// TIA Portal project "plc作业" (V15.1)

(* hardware
DEVICE "HMI_1"  KTP700 Basic PN
   slot 0: "HMI_1"  KTP700 Basic PN  6AV2 123-2GB03-0AX0  15.1.0.0
   slot 1: "HMI_RT_1"  KTP700 Basic PN  6AV2 123-2GB03-0AX0  15.1.0.0
   slot 5: "HMI_1.IE_CP_1"  PROFINET Interface  15.0.1.0
      slot 1: "PROFINET Interface_1"  PROFINET Interface
         slot 1: "Port_1"  Port
DEVICE "S7-1200 station_1"  S7-1200 Station
   slot 0: "Rack_0"  S7-1200 Rack  Rack  V1.0
   slot 1: "PLC_1"  CPU 1214C DC/DC/DC  6ES7 214-1AG40-0XB0  V4.2
*)

// ===== PLC "PLC_1"  CPU 1214C DC/DC/DC =====

VAR_GLOBAL   // PLC tag table "默认变量表"
   "Tag_1" AT %M500.0 : Bool;
   "Tag_2" AT %M500.1 : Bool;
   "Tag_3" AT %M500.2 : Bool;
   "Tag_22" AT %M501.0 : Bool;
   "Tag_23" AT %M501.1 : Bool;
   "Tag_24" AT %M501.2 : Bool;
   "Tag_25" AT %M500.5 : Bool;
   "Tag_26" AT %M500.6 : Bool;
   "Tag_27" AT %M500.7 : Bool;
END_VAR

VAR_GLOBAL   // PLC tag table "左车道检测"
   "使能信号" AT %I0.6 : Bool;
   "左车道入口计数" AT %I0.7 : Bool;
   "左车道出口计数" AT %I1.1 : Bool;
   "左车道计数清零" AT %I1.3 : Bool;
   "左车道封闭" AT %Q0.2 : Bool;
   "左车道堵塞" AT %Q0.3 : Bool;
   "左车道拥堵" AT %Q0.4 : Bool;
   "左车道畅通" AT %Q0.5 : Bool;
   "左车道hmi停止控制" AT %M2.0 : Bool;
   "左车道错误" AT %M2.1 : Bool;
END_VAR

VAR_GLOBAL   // PLC tag table "右车道"
   "右车道入口计数" AT %I1.0 : Bool;
   "右车道出口计数" AT %I1.2 : Bool;
   "右车道计数清零" AT %I1.4 : Bool;
   "右车道封闭" AT %Q0.6 : Bool;
   "右车道堵塞" AT %Q0.7 : Bool;
   "右车道拥堵" AT %Q1.0 : Bool;
   "右车道畅通" AT %Q1.1 : Bool;
   "右车道hmi停止控制" AT %M2.2 : Bool;
   "右车道错误" AT %M2.3 : Bool;
END_VAR

DATA_BLOCK "车辆检测_DB"   // DB1
{ S7_Optimized_Access := 'FALSE' }
VERSION : 0.1
// stored: InstanceOfName 车辆检测
"车辆检测"
BEGIN
   堵塞设定数量 := 15;
   拥堵设定数量 := 10;
END_DATA_BLOCK

DATA_BLOCK "车辆检测_DB_1"   // DB2
{ S7_Optimized_Access := 'FALSE' }
VERSION : 0.1
// stored: InstanceOfName 车辆检测
"车辆检测"
BEGIN
   堵塞设定数量 := 15;
   拥堵设定数量 := 10;
END_DATA_BLOCK

FUNCTION_BLOCK "车辆检测"   // FB1, LAD
{ S7_Optimized_Access := 'FALSE' }
VERSION : 0.1
   VAR_INPUT
      使能信号 : Bool;
      车道入口计数 : Bool;
      出口计数 : Bool;
      计数清零 : Bool;
      停止控制 : Bool;
   END_VAR
   VAR_OUTPUT
      封闭 : Bool;
      堵塞 : Bool;
      拥堵 : Bool;
      畅通 : Bool;
      错误 : Bool;
   END_VAR
   VAR_IN_OUT
      堵塞设定数量 : Int;
      拥堵设定数量 : Int;
      当前车辆数量 : Int;
      "step" : Bool;
   END_VAR
   VAR_TEMP   // added for the SCL form of the ladder/FBD networks
      _w1 : Bool;
      _w2 : Bool;
   END_VAR
BEGIN

REGION Network 1
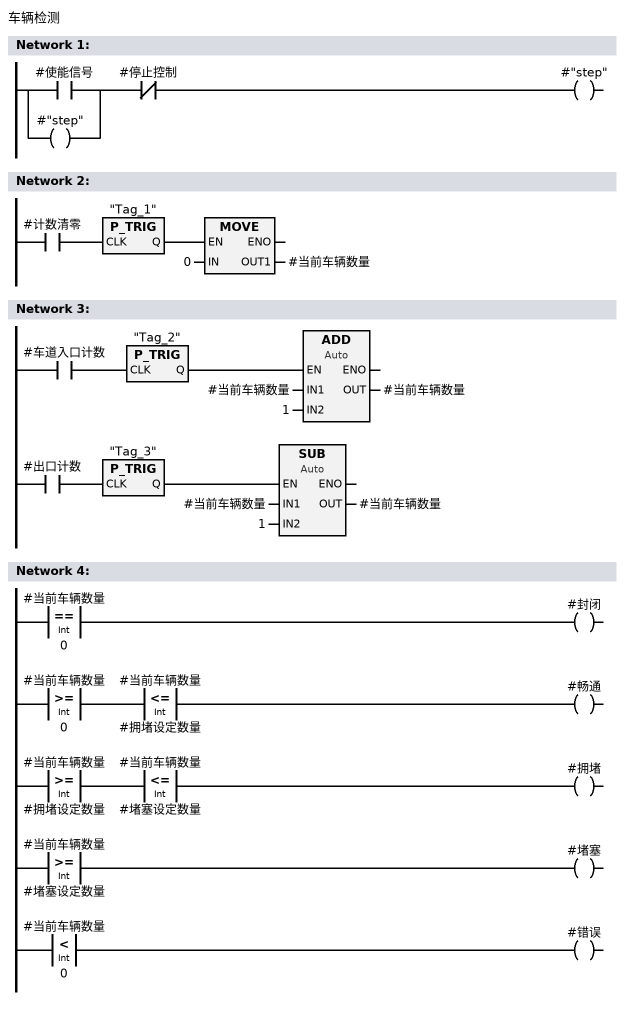
   RUNG wire#powerrail
      Contact( #使能信号 )
      wire#w1
      I_Contact( #停止控制 )
      Coil( #"step" )
   END_RUNG
   RUNG wire#powerrail
      Coil( #"step" )
   END_RUNG wire#w1
   // the same network as SCL:
   #"step" := TRUE;
   #"step" := (#使能信号 OR TRUE) AND NOT #停止控制;
END_REGION

REGION Network 2
   RUNG wire#powerrail
      Contact( #计数清零 )
      P_Trig( "Tag_1" )
      Move(in := 0, out1 => #当前车辆数量)
   END_RUNG
   // the same network as SCL:
   #_w1 := #计数清零 AND NOT "Tag_1";   // rising edge
   "Tag_1" := #计数清零;
   IF #_w1 THEN #当前车辆数量 := 0; END_IF;
END_REGION

REGION Network 3
   RUNG wire#powerrail
      Contact( #车道入口计数 )
      P_Trig( "Tag_2" )
      Add(in1 := #当前车辆数量, in2 := 1, out => #当前车辆数量)
   END_RUNG
   RUNG wire#powerrail
      Contact( #出口计数 )
      P_Trig( "Tag_3" )
      Sub(in1 := #当前车辆数量, in2 := 1, out => #当前车辆数量)
   END_RUNG
   // the same network as SCL:
   #_w1 := #车道入口计数 AND NOT "Tag_2";   // rising edge
   "Tag_2" := #车道入口计数;
   IF #_w1 THEN #当前车辆数量 := #当前车辆数量 + 1; END_IF;
   #_w2 := #出口计数 AND NOT "Tag_3";   // rising edge
   "Tag_3" := #出口计数;
   IF #_w2 THEN #当前车辆数量 := #当前车辆数量 - 1; END_IF;
END_REGION

REGION Network 4
   RUNG wire#powerrail
      { S7_Templates := "SrcType := Int" } EQ_Contact(in1 := #当前车辆数量, in2 := 0)
      Coil( #封闭 )
   END_RUNG
   RUNG wire#powerrail
      { S7_Templates := "SrcType := Int" } GE_Contact(in1 := #当前车辆数量, in2 := 0)
      { S7_Templates := "SrcType := Int" } LE_Contact(in1 := #当前车辆数量, in2 := #拥堵设定数量)
      Coil( #畅通 )
   END_RUNG
   RUNG wire#powerrail
      { S7_Templates := "SrcType := Int" } GE_Contact(in1 := #当前车辆数量, in2 := #拥堵设定数量)
      { S7_Templates := "SrcType := Int" } LE_Contact(in1 := #当前车辆数量, in2 := #堵塞设定数量)
      Coil( #拥堵 )
   END_RUNG
   RUNG wire#powerrail
      { S7_Templates := "SrcType := Int" } GE_Contact(in1 := #当前车辆数量, in2 := #堵塞设定数量)
      Coil( #堵塞 )
   END_RUNG
   RUNG wire#powerrail
      { S7_Templates := "SrcType := Int" } LT_Contact(in1 := #当前车辆数量, in2 := 0)
      Coil( #错误 )
   END_RUNG
   // the same network as SCL:
   #封闭 := #当前车辆数量 = 0;
   #畅通 := (#当前车辆数量 >= 0) AND (#当前车辆数量 <= #拥堵设定数量);
   #拥堵 := (#当前车辆数量 >= #拥堵设定数量) AND (#当前车辆数量 <= #堵塞设定数量);
   #堵塞 := #当前车辆数量 >= #堵塞设定数量;
   #错误 := #当前车辆数量 < 0;
END_REGION
END_FUNCTION_BLOCK

ORGANIZATION_BLOCK "Main"   // OB1, LAD, ProgramCycle
TITLE = "Main Program Sweep (Cycle)"
{ S7_Optimized_Access := 'TRUE' }
VERSION : 0.1
   VAR_INPUT
      Initial_Call : Bool;   // Initial call of this OB
      Remanence : Bool;   // =True, if remanent data are available
   END_VAR
   VAR_TEMP   // added for the SCL form of the ladder/FBD networks
      _w1 : Bool;
      _w2 : Bool;
      _w3 : Bool;
   END_VAR
BEGIN

REGION Network 1: 左车道
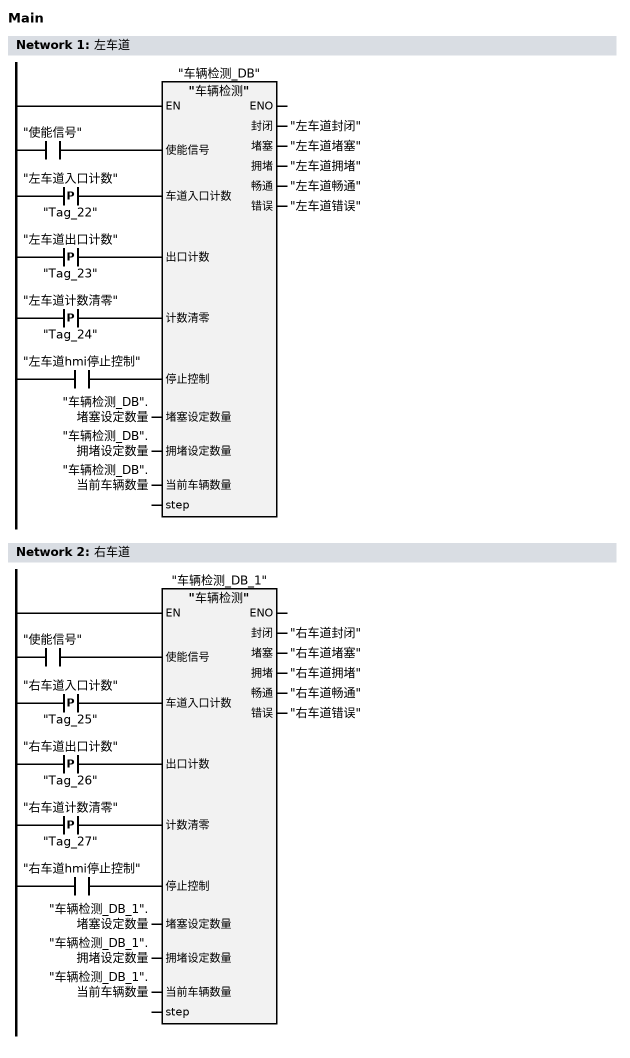
   RUNG wire#powerrail
      "车辆检测_DB"(使能信号 := wire#w1, 车道入口计数 := wire#w2, 出口计数 := wire#w3, 计数清零 := wire#w4, 停止控制 := wire#w5, 堵塞设定数量 := "车辆检测_DB".堵塞设定数量, 拥堵设定数量 := "车辆检测_DB".拥堵设定数量, 当前车辆数量 := "车辆检测_DB".当前车辆数量, "step" :=, 封闭 => "左车道封闭", 堵塞 => "左车道堵塞", 拥堵 => "左车道拥堵", 畅通 => "左车道畅通", 错误 => "左车道错误")
   END_RUNG
   RUNG wire#powerrail
      Contact( "使能信号" )
   END_RUNG wire#w1
   RUNG wire#powerrail
      P_Contact(operand := "左车道入口计数", bit := "Tag_22")
   END_RUNG wire#w2
   RUNG wire#powerrail
      P_Contact(operand := "左车道出口计数", bit := "Tag_23")
   END_RUNG wire#w3
   RUNG wire#powerrail
      P_Contact(operand := "左车道计数清零", bit := "Tag_24")
   END_RUNG wire#w4
   RUNG wire#powerrail
      Contact( "左车道hmi停止控制" )
   END_RUNG wire#w5
   // the same network as SCL:
   #_w1 := "左车道入口计数" AND NOT "Tag_22";   // rising edge of "左车道入口计数"
   "Tag_22" := "左车道入口计数";
   #_w2 := "左车道出口计数" AND NOT "Tag_23";   // rising edge of "左车道出口计数"
   "Tag_23" := "左车道出口计数";
   #_w3 := "左车道计数清零" AND NOT "Tag_24";   // rising edge of "左车道计数清零"
   "Tag_24" := "左车道计数清零";
   "车辆检测_DB"(使能信号 := "使能信号",   // "车辆检测"
             车道入口计数 := #_w1,
             出口计数 := #_w2,
             计数清零 := #_w3,
             停止控制 := "左车道hmi停止控制",
             堵塞设定数量 := "车辆检测_DB".堵塞设定数量,
             拥堵设定数量 := "车辆检测_DB".拥堵设定数量,
             当前车辆数量 := "车辆检测_DB".当前车辆数量,
             封闭 => "左车道封闭",
             堵塞 => "左车道堵塞",
             拥堵 => "左车道拥堵",
             畅通 => "左车道畅通",
             错误 => "左车道错误");
END_REGION

REGION Network 2: 右车道
   RUNG wire#powerrail
      "车辆检测_DB_1"(使能信号 := wire#w1, 车道入口计数 := wire#w2, 出口计数 := wire#w3, 计数清零 := wire#w4, 停止控制 := wire#w5, 堵塞设定数量 := "车辆检测_DB_1".堵塞设定数量, 拥堵设定数量 := "车辆检测_DB_1".拥堵设定数量, 当前车辆数量 := "车辆检测_DB_1".当前车辆数量, "step" :=, 封闭 => "右车道封闭", 堵塞 => "右车道堵塞", 拥堵 => "右车道拥堵", 畅通 => "右车道畅通", 错误 => "右车道错误")
   END_RUNG
   RUNG wire#powerrail
      Contact( "使能信号" )
   END_RUNG wire#w1
   RUNG wire#powerrail
      P_Contact(operand := "右车道入口计数", bit := "Tag_25")
   END_RUNG wire#w2
   RUNG wire#powerrail
      P_Contact(operand := "右车道出口计数", bit := "Tag_26")
   END_RUNG wire#w3
   RUNG wire#powerrail
      P_Contact(operand := "右车道计数清零", bit := "Tag_27")
   END_RUNG wire#w4
   RUNG wire#powerrail
      Contact( "右车道hmi停止控制" )
   END_RUNG wire#w5
   // the same network as SCL:
   #_w1 := "右车道入口计数" AND NOT "Tag_25";   // rising edge of "右车道入口计数"
   "Tag_25" := "右车道入口计数";
   #_w2 := "右车道出口计数" AND NOT "Tag_26";   // rising edge of "右车道出口计数"
   "Tag_26" := "右车道出口计数";
   #_w3 := "右车道计数清零" AND NOT "Tag_27";   // rising edge of "右车道计数清零"
   "Tag_27" := "右车道计数清零";
   "车辆检测_DB_1"(使能信号 := "使能信号",   // "车辆检测"
               车道入口计数 := #_w1,
               出口计数 := #_w2,
               计数清零 := #_w3,
               停止控制 := "右车道hmi停止控制",
               堵塞设定数量 := "车辆检测_DB_1".堵塞设定数量,
               拥堵设定数量 := "车辆检测_DB_1".拥堵设定数量,
               当前车辆数量 := "车辆检测_DB_1".当前车辆数量,
               封闭 => "右车道封闭",
               堵塞 => "右车道堵塞",
               拥堵 => "右车道拥堵",
               畅通 => "右车道畅通",
               错误 => "右车道错误");
END_REGION
END_ORGANIZATION_BLOCK

(* ===== HMI "HMI_RT_1" =====
system functions are stored by id; their names below are inferred from use
connection "Connection_1": ETHERNET, SMART_S7_1200_OMS
connection "HMI_连接_1": ETHERNET, SMART_S7_1200_OMS

HMI tags "默认变量表"
   "Tag_ScreenNumber" : UInt, internal
   "左车道畅通" : Bool = PLC 左车道畅通 AT %Q0.5, 1 s
   "左车道封闭" : Bool = PLC 左车道封闭 AT %Q0.2, 1 s
   "左车道堵塞" : Bool = PLC 左车道堵塞 AT %Q0.3, 1 s
   "左车道拥堵" : Bool = PLC 左车道拥堵 AT %Q0.4, 1 s
   "左车道错误" : Bool = PLC 左车道错误 AT %M2.1, 1 s
   "右车道封闭" : Bool = PLC 右车道封闭 AT %Q0.6, 1 s
   "右车道堵塞" : Bool = PLC 右车道堵塞 AT %Q0.7, 1 s
   "右车道拥堵" : Bool = PLC 右车道拥堵 AT %Q1.0, 1 s
   "右车道畅通" : Bool = PLC 右车道畅通 AT %Q1.1, 1 s
   "右车道错误" : Bool = PLC 右车道错误 AT %M2.3, 1 s
   "车辆检测_DB_当前车辆数量" : Int = PLC 车辆检测_DB.当前车辆数量 AT %DB1.DBW8, 1 s
   "车辆检测_DB_1_当前车辆数量" : Int = PLC 车辆检测_DB_1.当前车辆数量 AT %DB2.DBW8, 1 s
   "左车道hmi停止控制" : Bool = PLC 左车道hmi停止控制 AT %M2.0, 1 s
   "右车道hmi停止控制" : Bool = PLC 右车道hmi停止控制 AT %M2.2, 1 s

Template "模板_1" 800x480
   Button "退出" at 714,429 size 71x50; TextOff '退出'; PictureOff "ExitRuntime_KTP700_Basic_PN_TR"; PictureOn "ExitRuntime_KTP700_Basic_PN_TR"
      on Release: StopRuntime(0)
   Button "Template_Button" at 614,429 size 71x50; TextOff 'Text'
   Button "Template_Button_1" at 514,429 size 71x50; TextOff 'Text'
   Button "Template_Button_2" at 414,429 size 71x50; TextOff 'Text'
   Button "Template_Button_3" at 314,429 size 71x50; TextOff 'Text'
   Button "Template_Button_4" at 214,429 size 71x50; TextOff 'Text'
   Button "Template_Button_5" at 114,429 size 71x50; TextOff 'Text'
   Button "起始画面" at 14,429 size 71x50; TextOff '起始画面'; PictureOff "NavigateHome_KTP700_Basic_PN_TR"; PictureOn "NavigateHome_KTP700_Basic_PN_TR"
      on Release: ActivateScreen("根画面", 0)
   SymbolicIOField "Symbolic_IO_Field_Screen" at 93,9 size 600x33; TextOff '0'; TextOn '1'; TextList "TextList_ScreenNames"
      ProcessValue <- "Tag_ScreenNumber"
      on Change: ActivateScreenByNumber("Tag_ScreenNumber", 0)
   DateTimeField "HmiScreenItemData" at 695,25 size 105x25
   DateTimeField "HmiScreenItemData_1" at 695,0 size 105x25
   GraphicView "Logo" at 0,0 size 91x51; Picture "HMI_1 的 Logo"

screen "根画面" 800x480, template "模板_1"
   on GenerateScreen: SetTag("Tag_ScreenNumber", 1)
   Visibility <- "车辆检测_DB_当前车辆数量"
   Circle "圆_1" at 50,86 size 48x48
      Appearance <- "左车道封闭"
   Circle "圆_2" at 142,82 size 48x48
      Appearance <- "左车道堵塞"
   Circle "圆_3" at 237,86 size 48x48
      Appearance <- "左车道拥堵"
   Circle "圆_4" at 341,86 size 48x48
      Appearance <- "左车道畅通"
   Circle "圆_5" at 452,86 size 48x48
      Appearance <- "左车道错误"
   Circle "圆_6" at 50,182 size 48x48
      Appearance <- "右车道封闭"
   Circle "圆_7" at 142,182 size 48x48
      Appearance <- "右车道堵塞"
   Circle "圆_8" at 236,183 size 48x48
      Appearance <- "右车道拥堵"
   Circle "圆_9" at 341,183 size 48x48
      Appearance <- "右车道畅通"
   Circle "圆_10" at 452,183 size 48x48
      Appearance <- "右车道错误"
   Button "按钮_1" at 116,295 size 96x32; TextOff '左停止'
      on Activate: InvertBit("左车道hmi停止控制")
   Button "按钮_2" at 116,372 size 96x32; TextOff '右停止'
      on Activate: InvertBit("右车道hmi停止控制")
   IOField "I/O 域_1" at 624,295 size 96x32; FormatPattern s99999
      ProcessValue <- "车辆检测_DB_当前车辆数量"
   IOField "I/O 域_2" at 627,372 size 96x32; FormatPattern s99999
      ProcessValue <- "车辆检测_DB_1_当前车辆数量"
   TextField "文本域_1" at 488,295 size 124x20; Text '左车道当前数量'
   TextField "文本域_2" at 482,372 size 124x20; Text '右车道当前数量'
   TextField "文本域_3" at 54,152 size 39x20; Text '封闭'
   TextField "文本域_4" at 163,163 size 14x20; Text 'Text'
   TextField "文本域_5" at 8,8 size 41x20; Text 'Text'
   TextField "文本域_6" at 139,152 size 39x20; Text '堵塞'
   TextField "文本域_7" at 232,156 size 39x20; Text '拥堵'
   TextField "文本域_8" at 341,152 size 39x20; Text '畅通'
   TextField "文本域_9" at 452,152 size 39x20; Text '停止'
   TextField "文本域_10" at 50,245 size 39x20; Text '封闭'
   TextField "文本域_11" at 136,247 size 39x20; Text '堵塞'
   TextField "文本域_12" at 234,247 size 39x20; Text '拥堵'
   TextField "文本域_13" at 340,247 size 39x20; Text '畅通'
   TextField "文本域_14" at 458,247 size 39x20; Text '停止'
   TextField "文本域_15" at 535,97 size 56x20; Text '左车道'
   TextField "文本域_16" at 536,188 size 56x20; Text '右车道'
*)